RoboDK station: Robodk Palletising system good.rdk

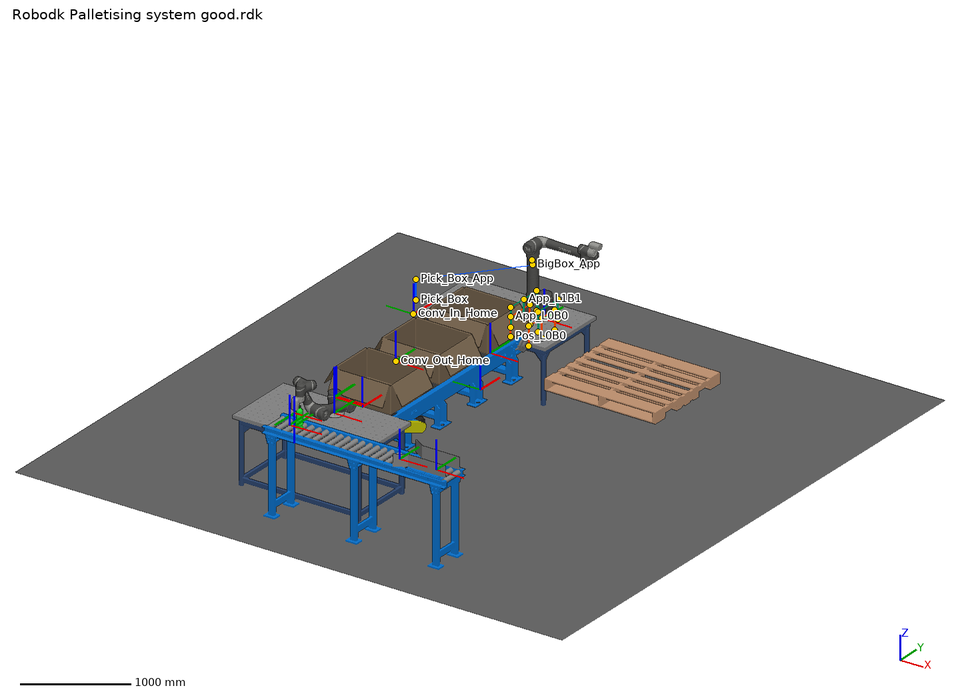
[picture v0: the station drawn from its stored meshes, robots at their saved joint values, targets as dots, program paths as lines]
Station Robodk Palletising system good (saved by RoboDK 5.5.3). Poses are relative to the parent item; angles as X-Y-Z fixed-axis rotations.
Station parameters (name, value as stored): TAGS, ['Packaging', 'Material Handling', 'Conveyor']
  - frame RoboDK RDK-1440 Base at (0, 0, 290) mm, rotated rx 0 ry 0 rz 90 deg
  - frame Conveyor Belt Base_Out at (-1180, 360, 105) mm
    - target Conv_Out_Home (Cartesian target) at (0, 0, 0) mm; joints [0, 0, 0, 0, 0, 0]
    - target BigBox_App (Cartesian target) at (1187.6, 447.36, 1114.86) mm, rotated rx -180 ry 0 rz -90 deg; joints [0.182, 1.544, 6.858, 0, 81.598, 0.182]
    - frame Belt_ConvWide Base at (1000, -1950, 600) mm, rotated rx 0 ry 0 rz 90 deg
      - robot Belt_ConvWide: 1 axes
          modified DH rows (alpha deg, a mm, theta deg, d mm): 0, 0, 0, 0 linear
          base shift (0, 0, 0) mm, rotated rx 0 ry 90 rz 0 deg
          joint limits [-200000] to [200000]; home [0]; saved at [0]
        - frame Frame_WideConv_Box at (30, 310, 10) mm, rotated rx 0 ry 0 rz -90 deg
          - object Box_24X20 at (0, -30, 0) mm, rotated rx 0 ry 0 rz -90 deg, size 750 x 855.1 x 305.2 mm, geometry from Big_Box.stl
          - object Box_24X20 at (0, 730, 0) mm, rotated rx 0 ry 0 rz -90 deg, size 750 x 855.1 x 305.2 mm, geometry from Big_Box.stl
          - object Box_24X20 at (0, 1490, 0) mm, rotated rx 0 ry 0 rz -90 deg, size 750 x 855.1 x 305.2 mm, geometry from Big_Box.stl
      - frame NewBox_24X20_Init at (0, 310, 10) mm, rotated rx 0 ry 0 rz -90 deg
        - object Box_24X20_Ref at (0, 0, 0) mm, rotated rx 0 ry 0 rz -90 deg, size 750 x 855.1 x 305.2 mm, geometry from Big_Box.stl
        - object Box_24X20_Ref at (0, 760, 0) mm, rotated rx 0 ry 0 rz -90 deg, size 750 x 855.1 x 305.2 mm, geometry from Big_Box.stl
        - object Box_24X20_Ref at (0, 1520, 0) mm, rotated rx 0 ry 0 rz -90 deg, size 750 x 855.1 x 305.2 mm, geometry from Big_Box.stl
      - frame NewBox_24X20_Ref at (0, 310, 10) mm, rotated rx 0 ry 0 rz -90 deg
        - object Box_24X20_Ref at (0, 0, 0) mm, rotated rx 0 ry 0 rz -90 deg, size 750 x 855.1 x 305.2 mm, geometry from Big_Box.stl
    - object Floor at (1380, -650, -105) mm, rotated rx 0 ry 0 rz 180 deg, size 6000 x 6000 x 0 mm, geometry from Floor.sld
    - frame PalletizingBaseFrame at (925, 166, 270) mm
      - target Palletizing_TargetConfig (Cartesian target) at (262.6, 277.36, 894.86) mm, rotated rx -180 ry 0 rz -90 deg; joints [57.652, 32.581, -14.377, 0, 71.796, 57.652]
      - folder Palletizing Data
        - folder Layer 0
          - target App_L0B0 (Cartesian target) at (108.4, 155.99, 333.74) mm, rotated rx 180 ry 0 rz -90 deg; joints [13.917, 14.572, 47.385, 0, 28.043, 13.917]
          - target Pos_L0B0 (Cartesian target) at (108.4, 155.99, 133.74) mm, rotated rx 180 ry 0 rz -90 deg; joints [13.917, 33.728, 48.412, 0, 7.86, 13.917]
          - target App_L0B1 (Cartesian target) at (108.4, 461.07, 333.74) mm, rotated rx 180 ry 0 rz -90 deg; joints [9.488, 33.379, 17.195, 0, 39.426, 9.488]
          - target Pos_L0B1 (Cartesian target) at (108.4, 461.07, 133.74) mm, rotated rx 180 ry 0 rz -90 deg; joints [9.488, 46.005, 18.009, 0, 25.986, 9.488]
          - target App_L0B2 (Cartesian target) at (355, 91.63, 333.74) mm, rotated rx 180 ry 0 rz 179.86 deg; joints [-4.557, 13.171, 49.353, 0, 27.475, 85.58]
          - target Pos_L0B2 (Cartesian target) at (355, 91.63, 133.74) mm, rotated rx 180 ry 0 rz 179.86 deg; joints [-4.557, 33.053, 50.41, 0, 6.538, 85.58]
          - target App_L0B3 (Cartesian target) at (355, 295.97, 333.74) mm, rotated rx 180 ry 0 rz 179.86 deg; joints [-3.441, 26.054, 29.653, 0, 34.293, 86.696]
          - target Pos_L0B3 (Cartesian target) at (355, 295.97, 133.74) mm, rotated rx 180 ry 0 rz 179.86 deg; joints [-3.441, 40.633, 30.513, 0, 18.854, 86.696]
          - target App_L0B4 (Cartesian target) at (355, 498.19, 333.74) mm, rotated rx 180 ry 0 rz 179.86 deg; joints [-2.769, 38.994, 7.222, 0, 43.784, 87.368]
          - target Pos_L0B4 (Cartesian target) at (355, 498.19, 133.74) mm, rotated rx 180 ry 0 rz 179.86 deg; joints [-2.769, 50.475, 8.028, 0, 31.497, 87.368]
        - folder Layer 1
          - target App_L1B0 (Cartesian target) at (155.97, 91.63, 467.48) mm, rotated rx 180 ry 0 rz 179.86 deg; joints [13.353, 4.2, 43.75, 0, 42.051, 103.49]
          - target Pos_L1B0 (Cartesian target) at (155.97, 91.63, 267.48) mm, rotated rx 180 ry 0 rz 179.86 deg; joints [13.353, 20.146, 48.998, 0, 20.857, 103.49]
          - target App_L1B1 (Cartesian target) at (155.97, 295.63, 467.48) mm, rotated rx 180 ry 0 rz 179.86 deg; joints [10.157, 19.153, 24.952, 0, 45.895, 100.293]
          - target Pos_L1B1 (Cartesian target) at (155.97, 295.63, 267.48) mm, rotated rx 180 ry 0 rz 179.86 deg; joints [10.157, 31.187, 29.359, 0, 29.454, 100.293]
          - target App_L1B2 (Cartesian target) at (155.97, 499.63, 467.48) mm, rotated rx 180 ry 0 rz 179.86 deg; joints [8.186, 33.828, 2.5, 0, 53.672, 98.323]
          - target Pos_L1B2 (Cartesian target) at (155.97, 499.63, 267.48) mm, rotated rx 180 ry 0 rz 179.86 deg; joints [8.186, 43.195, 6.716, 0, 40.09, 98.323]
          - target App_L1B3 (Cartesian target) at (413.47, 155.99, 467.48) mm, rotated rx 180 ry 0 rz -90 deg; joints [-13.221, 4.519, 43.398, 0, 42.083, -13.221]
          - target Pos_L1B3 (Cartesian target) at (413.47, 155.99, 267.48) mm, rotated rx 180 ry 0 rz -90 deg; joints [-13.221, 20.367, 48.622, 0, 21.011, -13.221]
          - target App_L1B4 (Cartesian target) at (413.47, 461.07, 467.48) mm, rotated rx 180 ry 0 rz -90 deg; joints [-9.003, 26.619, 13.952, 0, 49.429, -9.003]
          - target Pos_L1B4 (Cartesian target) at (413.47, 461.07, 267.48) mm, rotated rx 180 ry 0 rz -90 deg; joints [-9.003, 37.176, 18.179, 0, 34.645, -9.003]
  - frame Conveyor Belt Base_In at (-690, -60, 880) mm, rotated rx 0 ry 0 rz 90 deg
    - target Conv_In_Home (Cartesian target) at (0, 0, 0) mm; joints [0, 0, 0, 0, 0, 0]
    - target Pick_Box (Cartesian target) at (25.04, -7.77, 134.86) mm, rotated rx 180 ry 0 rz -180 deg; joints [96.997, -1.128, 27.465, 0, 63.663, 96.997]
    - target Pick_Box_App (Cartesian target) at (25.04, -7.77, 339.86) mm, rotated rx -180 ry 0 rz -180 deg; joints [96.997, -3.507, 11.821, 0, 81.687, 96.997]
    - frame Roller_Conv Base at (-2500, -2000, 0) mm, rotated rx 0 ry 0 rz -90 deg
      - robot Roller_Conv: 1 axes
          modified DH rows (alpha deg, a mm, theta deg, d mm): 0, 0, 0, 0 linear
          base shift (0, 0, 0) mm, rotated rx 0 ry 90 rz 0 deg
          joint limits [-200000] to [200000]; home [0]; saved at [-400]
        - frame Frame_Conv_Box at (0, 0, 0) mm
      - frame New_Box_12X7 at (-1560, 0, 0) mm
        - object Box 12X7_Ref at (-120, 100, 0) mm, rotated rx 0 ry 0 rz -90 deg, size 199 x 305.1 x 133.7 mm, geometry from Box 24x16 closed.step
        - frame Box 12X7_FrameRef at (0, 0, 135) mm, rotated rx 180 ry 0 rz 0 deg
      - frame New_Box_12X7_INIT at (-1610, 0, 0) mm
        - object Box 12X7_Ref at (550, 100, 0) mm, rotated rx 0 ry 0 rz -90 deg, size 199 x 305.1 x 133.7 mm, geometry from Box 24x16 closed.step
        - object Box 12X7_Ref at (860, 100, 0) mm, rotated rx 0 ry 0 rz -90 deg, size 199 x 305.1 x 133.7 mm, geometry from Box 24x16 closed.step
        - object Box 12X7_Ref at (1170, 100, 0) mm, rotated rx 0 ry 0 rz -90 deg, size 199 x 305.1 x 133.7 mm, geometry from Box 24x16 closed.step
        - object Box 12X7_Ref1 at (1480, 100, 0) mm, rotated rx 0 ry 0 rz -90 deg, size 199 x 305.1 x 133.7 mm, geometry from Box 24x16 closed.step
        - object Box 12X7_Ref at (240, 100, 0) mm, rotated rx 0 ry 0 rz -90 deg, size 199 x 305.1 x 133.7 mm, geometry from Box 24x16 closed.step
  - folder Python
    - Python program Reset_Conveyor (listed below)
    - Python program New_Box_24X16 (listed below)
    - Python program Reset_WideConveyor (listed below)
    - Python program New_Box_24X20 (listed below)
    - Python program Clear_Tool (listed below)
  - program PickBox (9 instructions, listed below)
  - program DropBox (1 instructions, listed below)
  - program RunConv_Out (4 instructions, listed below)
  - program RESET (5 instructions, listed below)
  - item type 20 Palletizing Settings: svg | Palletizing Plugin | PalletizingBaseFrame | Box 12X7_Ref1 | Box 12X7_Ref1 | Box 12X7_Ref1 | Box 12X7_Ref1 | Palletizing_TargetConfig | Depalletizing | Pos_L%1_B%2 | App_L%1_B%2 | Layer_%LAYER_NUM%_End | Ret_L%1_B%2_W%3 | %PROJECT_NAME%_L%LAYER_NUM% | %PROJECT_NAME%_L%LAYER_NUM%_B%BOX_NUM%
  - folder Palletizing
    - program Palletizing_Main (5 instructions, listed below)
    - program Palletizing_L0 (36 instructions, listed below)
    - program Palletizing_L1 (36 instructions, listed below)
  - program Main (2 instructions, listed below)
  - frame Omron TM5-700 Base at (-200, -2000, 800) mm
    - robot Omron TM5-700: 6 axes, payload 6 kg, reach 700 mm, repeatability 0.1 mm, weight 25 kg
        modified DH rows (alpha deg, a mm, theta deg, d mm): 0, 0, 0, 145.2; 90, 0, 90, 0; 0, 329, 0, 0; 0, 311, -90, 122.3; -90, 0, 0, 106.5; 90, 0, 180, 114.15
        joint limits [-270, -180, -155, -180, -180, -270] to [270, 180, 155, 180, 180, 270]; home [0, 0, 90, -90, 90, 0]; saved at [79.622, -84.489, 62.67, -67.315, -93.132, -10.928]
      - tool Tool 1, TCP at (0, 0, 150) mm
  - frame Omron TM12 Base at (0, 1000, 600) mm
    - robot Omron TM12: 6 axes, payload 12 kg, reach 1300 mm, repeatability 0.1 mm, weight 33.3 kg
        modified DH rows (alpha deg, a mm, theta deg, d mm): 0, 0, 0, 165.2; 90, 0, 90, 0; 0, 636.1, 0, 0; 0, 557.9, -90, 156.3; -90, 0, 0, 106; 90, 0, 180, 113.15
        joint limits [-270, -180, -166, -180, -180, -270] to [270, 180, 166, 180, 180, 270]; home [0, 0, 90, -90, 90, 0]; saved at [0, 0, 90, -90, 90, 0]
  - object Pallet 40inx48in at (700, 0, 600) mm, size 1219.2 x 1016 x 114.3 mm, geometry from AR3.step
  - object Table 1400x800x800mm at (-700, 900, 610) mm, size 1420 x 820 x 800 mm, geometry from Table-1400x800x800mm.sld
  - object Table 1400x800x800mm at (-700, -2000, 710) mm, size 1420 x 820 x 800 mm, geometry from Table-1400x800x800mm.sld
  - object Coffee 1 at (-200, -2550, 870) mm, size 71.4 x 71.4 x 225.2 mm, geometry from moutaindew.STEP
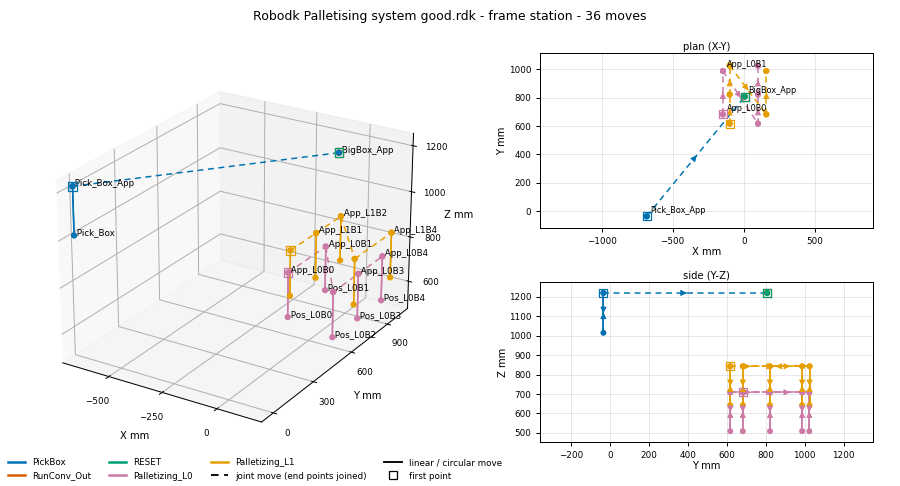
[picture p0: tool path of Robodk Palletising system good.rdk in frame station, 36 of 36 moves have a stored position in this frame; points joined in program order, loops and branches not executed]

--- Python program Reset_Conveyor ---
# Type help("robolink") or help("robodk") for more information
# Press F5 to run the script
# Documentation: https://robodk.com/doc/en/RoboDK-API.html
# Reference:     https://robodk.com/doc/en/PythonAPI/index.html
# Note: It is not required to keep a copy of this file, your python script is saved with the station
from robolink import *    # RoboDK API
from robodk import *      # Robot toolbox
RDK = Robolink()

#----- CONSTANT -----
CONV_FRAME_NAME = 'Frame_Conv_Box'
NEW_REF_OBJECT_NAME = 'Box 12X7_Ref' #Name of the ref object to copy
NEW_OBJECT_NAME = 'Box_12X7' #Name of the new object created
REFERENCE_FRAME = 'Frame_Conv_Box' #Name of the frame the object will move to
REFERENCE_FRAME_REF = 'New_Box_12X7_INIT'


#----- PROGRAM -----
frame = RDK.Item(CONV_FRAME_NAME,ITEM_TYPE_FRAME)

if frame.Valid():
    for item in frame.Childs():
        if item.Type() == ITEM_TYPE_OBJECT:
            item.Delete()

#This program reinitialize every mechanisms in the list to position 0
MECHANISM_LIST = ["Roller_Conv"]

for i in range(len(MECHANISM_LIST)):
    MECHANISM_NAME=MECHANISM_LIST[i]
    mechanism = RDK.Item(MECHANISM_NAME,itemtype=ITEM_TYPE_ROBOT)
    if mechanism.Valid():
        mechanism.setJoints([0])

#------- Program ------
frame = RDK.Item(REFERENCE_FRAME, ITEM_TYPE_FRAME)
frame_ref = RDK.Item(REFERENCE_FRAME_REF, ITEM_TYPE_FRAME)
ref_obj = RDK.Item(NEW_REF_OBJECT_NAME, ITEM_TYPE_OBJECT)

RDK.Render(False)

for item in frame_ref.Childs():
    if frame.Valid() and  ref_obj.Valid():
        item.Copy()
        new_obj = RDK.Paste()
        new_obj.setVisible(False)
        new_obj.setName(NEW_OBJECT_NAME)
        new_obj.setParent(frame_ref)
        RDK.Update()
        new_obj.setParentStatic(frame)
        new_obj.setVisible(True)
RDK.Render(True)

--- Python program New_Box_24X16 ---
# Type help("robolink") or help("robodk") for more information
# Press F5 to run the script
# Documentation: https://robodk.com/doc/en/RoboDK-API.html
# Reference:     https://robodk.com/doc/en/PythonAPI/index.html
# Note: It is not required to keep a copy of this file, your python script is saved with the station
from robolink import *    # RoboDK API
from robodk import *      # Robot toolbox
RDK = Robolink()



#----- Constante -----
NEW_REF_OBJECT_NAME = 'Box 12X7_Ref' #Name of the ref object to copy
NEW_OBJECT_NAME = 'Box_12X7' #Name of the new object created
REFERENCE_FRAME = 'Frame_Conv_Box' #Name of the frame the object will move to
REFERENCE_FRAME_REF = 'New_Box_12X7'
MECHANISM_NAME = 'Roller_Conv'
PART_TRAVEL_MM = 310 #Travel for each box


#------- Program ------
frame = RDK.Item(REFERENCE_FRAME, ITEM_TYPE_FRAME)
frame_ref = RDK.Item(REFERENCE_FRAME_REF, ITEM_TYPE_FRAME)
ref_obj = RDK.Item(NEW_REF_OBJECT_NAME, ITEM_TYPE_OBJECT)

#RDK.Render(False)
if frame.Valid() and  ref_obj.Valid():
    ref_obj.Copy()
    new_obj = RDK.Paste()
    new_obj.setVisible(False)
    new_obj.setName(NEW_OBJECT_NAME)
    new_obj.setParent(frame_ref)
    RDK.Update()
    new_obj.setParentStatic(frame)
    new_obj.setVisible(True)
#RDK.Render(True)


mechanism = RDK.Item(MECHANISM_NAME,itemtype=ITEM_TYPE_ROBOT)

if mechanism.Valid():
    mechanism.MoveJ(mechanism.Joints() + PART_TRAVEL_MM)

--- Python program Reset_WideConveyor ---
# Type help("robolink") or help("robodk") for more information
# Press F5 to run the script
# Documentation: https://robodk.com/doc/en/RoboDK-API.html
# Reference:     https://robodk.com/doc/en/PythonAPI/index.html
# Note: It is not required to keep a copy of this file, your python script is saved with the station
from robolink import *    # RoboDK API
from robodk import *      # Robot toolbox
RDK = Robolink()

#----- CONSTANT -----
CONV_FRAME_NAME = 'Frame_WideConv_Box'
NEW_REF_OBJECT_NAME = 'Box_24X20_Ref' #Name of the ref object to copy
NEW_OBJECT_NAME = 'Box_24X20' #Name of the new object created
REFERENCE_FRAME = 'Frame_WideConv_Box' #Name of the frame the object will move to
REFERENCE_FRAME_REF = 'NewBox_24X20_Init'

#This program reinitialize every mechanisms in the list to position 0
MECHANISM_LIST = ["Belt_ConvWide"]


#----- PROGRAM -----
frame = RDK.Item(CONV_FRAME_NAME,ITEM_TYPE_FRAME)

if frame.Valid():
    for item in frame.Childs():
        if item.Type() == ITEM_TYPE_OBJECT:
            item.Delete()



for i in range(len(MECHANISM_LIST)):
    MECHANISM_NAME=MECHANISM_LIST[i]
    mechanism = RDK.Item(MECHANISM_NAME,itemtype=ITEM_TYPE_ROBOT)
    if mechanism.Valid():
        mechanism.setJoints([0])

#------- Program ------
frame = RDK.Item(REFERENCE_FRAME, ITEM_TYPE_FRAME)
frame_ref = RDK.Item(REFERENCE_FRAME_REF, ITEM_TYPE_FRAME)
ref_obj = RDK.Item(NEW_REF_OBJECT_NAME, ITEM_TYPE_OBJECT)

RDK.Render(False)

for item in frame_ref.Childs():
    if frame.Valid() and  ref_obj.Valid():
        item.Copy()
        new_obj = RDK.Paste()
        new_obj.setVisible(False)
        new_obj.setName(NEW_OBJECT_NAME)
        new_obj.setParent(frame_ref)
        RDK.Update()
        new_obj.setParentStatic(frame)
        new_obj.setVisible(True)
RDK.Render(True)

--- Python program New_Box_24X20 ---
# Type help("robolink") or help("robodk") for more information
# Press F5 to run the script
# Documentation: https://robodk.com/doc/en/RoboDK-API.html
# Reference:     https://robodk.com/doc/en/PythonAPI/index.html
# Note: It is not required to keep a copy of this file, your python script is saved with the station
from robolink import *    # RoboDK API
from robodk import *      # Robot toolbox
RDK = Robolink()


#----- Constante -----
NEW_REF_OBJECT_NAME = 'Box_24X20_Ref' #Name of the ref object to copy
NEW_OBJECT_NAME = 'Box_24X20' #Name of the new object created
REFERENCE_FRAME = 'Frame_WideConv_Box' #Name of the frame the object will move to
REFERENCE_FRAME_REF = 'NewBox_24X20_Ref'
MECHANISM_NAME = 'Belt_ConvWide'
PART_TRAVEL_MM = 760 #Travel for each box


#------- Program ------
frame = RDK.Item(REFERENCE_FRAME, ITEM_TYPE_FRAME)
frame_ref = RDK.Item(REFERENCE_FRAME_REF, ITEM_TYPE_FRAME)
ref_obj = RDK.Item(NEW_REF_OBJECT_NAME, ITEM_TYPE_OBJECT)


#MOVE CONVEYOR

mechanism = RDK.Item(MECHANISM_NAME,itemtype=ITEM_TYPE_ROBOT)

if mechanism.Valid():
    mechanism.MoveJ(mechanism.Joints() + PART_TRAVEL_MM)

#CREATE NEW BOX

RDK.Render(False)
if frame.Valid() and  ref_obj.Valid():
    ref_obj.Copy()
    new_obj = RDK.Paste()
    new_obj.setVisible(False)
    new_obj.setName(NEW_OBJECT_NAME)
    new_obj.setParent(frame_ref)
    RDK.Update()
    new_obj.setParentStatic(frame)
    new_obj.setVisible(True)
RDK.Render(True)

#DELETE LAST BOX


#Declaration of the child frames
frame = frame.Childs()


for item in frame:
    #print(item.PoseAbs()) #If you want to see the Abs pos matrix of the object
    if item.PoseAbs()[0,3] > 1660: #[1,3] refer to line 0 column 3 in the pos matrix, so the Y position
        item.Delete()

--- Python program Clear_Tool ---
# Type help("robolink") or help("robodk") for more information
# Press F5 to run the script
# Documentation: https://robodk.com/doc/en/RoboDK-API.html
# Reference:     https://robodk.com/doc/en/PythonAPI/index.html
# Note: It is not required to keep a copy of this file, your python script is saved with the station
from robolink import *    # RoboDK API
from robodk import *      # Robot toolbox
RDK = Robolink()

#----- CONSTANT -----
TOOL_NAME = 'Gripper'

#----- PROGRAM -----
tool = RDK.Item(TOOL_NAME,ITEM_TYPE_TOOL)

if tool.Valid():
    for item in tool.Childs():
        if item.Type() == ITEM_TYPE_OBJECT:
            item.Delete()

--- program PickBox ---
  Set Ref.: Conveyor Belt Base_In
  Set Tool: Gripper at (-50, -10, 105) mm
  MoveJ (Pick_Box_App)
  MoveL (Pick_Box)
  Attach to Gripper
  MoveL (Pick_Box_App)
  Run New_Box_24X16
  Set Ref.: Conveyor Belt Base_Out
  MoveJ (BigBox_App)

--- program DropBox ---
  Detach from Gripper

--- program RunConv_Out ---
  Set Ref.: Conveyor Belt Base_Out
  Set Tool: Gripper at (-50, -10, 105) mm
  MoveJ (BigBox_App)
  Call New_Box_24X20

--- program RESET ---
  Call Reset_Conveyor
  Call Reset_WideConveyor
  Call Clear_Tool
  Set Ref.: Conveyor Belt Base_Out
  MoveJ (BigBox_App)

--- program Palletizing_Main ---
  Set Ref.: PalletizingBaseFrame
  Set Tool: Gripper at (-50, -10, 105) mm
  Call Palletizing_L0
  Call Palletizing_L1
  Call RunConv_Out

--- program Palletizing_L0 ---
  Set Ref.: PalletizingBaseFrame
  Call PickBox
  Set Ref.: PalletizingBaseFrame
  MoveJ (App_L0B0)
  MoveL (Pos_L0B0)
  Call DropBox
  Set Ref.: PalletizingBaseFrame
  MoveL (App_L0B0)
  Call PickBox
  Set Ref.: PalletizingBaseFrame
  MoveJ (App_L0B1)
  MoveL (Pos_L0B1)
  Call DropBox
  Set Ref.: PalletizingBaseFrame
  MoveL (App_L0B1)
  Call PickBox
  Set Ref.: PalletizingBaseFrame
  MoveJ (App_L0B2)
  MoveL (Pos_L0B2)
  Call DropBox
  Set Ref.: PalletizingBaseFrame
  MoveL (App_L0B2)
  Call PickBox
  Set Ref.: PalletizingBaseFrame
  MoveJ (App_L0B3)
  MoveL (Pos_L0B3)
  Call DropBox
  Set Ref.: PalletizingBaseFrame
  MoveL (App_L0B3)
  Call PickBox
  Set Ref.: PalletizingBaseFrame
  MoveJ (App_L0B4)
  MoveL (Pos_L0B4)
  Call DropBox
  Set Ref.: PalletizingBaseFrame
  MoveL (App_L0B4)

--- program Palletizing_L1 ---
  Set Ref.: PalletizingBaseFrame
  Call PickBox
  Set Ref.: PalletizingBaseFrame
  MoveJ (App_L1B0)
  MoveL (Pos_L1B0)
  Call DropBox
  Set Ref.: PalletizingBaseFrame
  MoveL (App_L1B0)
  Call PickBox
  Set Ref.: PalletizingBaseFrame
  MoveJ (App_L1B1)
  MoveL (Pos_L1B1)
  Call DropBox
  Set Ref.: PalletizingBaseFrame
  MoveL (App_L1B1)
  Call PickBox
  Set Ref.: PalletizingBaseFrame
  MoveJ (App_L1B2)
  MoveL (Pos_L1B2)
  Call DropBox
  Set Ref.: PalletizingBaseFrame
  MoveL (App_L1B2)
  Call PickBox
  Set Ref.: PalletizingBaseFrame
  MoveJ (App_L1B3)
  MoveL (Pos_L1B3)
  Call DropBox
  Set Ref.: PalletizingBaseFrame
  MoveL (App_L1B3)
  Call PickBox
  Set Ref.: PalletizingBaseFrame
  MoveJ (App_L1B4)
  MoveL (Pos_L1B4)
  Call DropBox
  Set Ref.: PalletizingBaseFrame
  MoveL (App_L1B4)

--- program Main ---
  Call RESET
  Call Palletizing_Main
